FUNCTION_BLOCK FB_ROB_MANIP EXTENDS FB_ROB IMPLEMENTS ITF_2_6AxisRobot



VAR_OUTPUT

END_VAR
VAR

	tcppos, tcpvel : stPose3D;
	jointpos, jointvel: stJoint6;
	currFrame: stFrame;
	currTool: FB_Tool;

END_VAR

//State Machine

{warning 'Add method implementation '}
METHOD M_Home : BOOL
END_METHOD

{warning 'Add method implementation '}
METHOD M_SwitchTool : UINT
VAR_INPUT
	tool	: FB_Tool;
END_VAR
END_METHOD

{warning 'Add method implementation '}
METHOD MC_MoveAxesAbsolute : BOOL
VAR_INPUT
	target	: stTarget3D;
END_VAR
IF _state=eState.Active THEN
// 	P_TargetReached:=FALSE;
END_IF
END_METHOD

{warning 'Add method implementation '}
METHOD MC_MoveAxesRelative : BOOL
VAR_INPUT
	axes	: ARRAY [1..6] OF FB_Axis;
	offsets	: ARRAY [1..6] OF REAL;
END_VAR
END_METHOD

{warning 'Add method implementation '}
METHOD MC_MoveLinearAbsolute : BOOL
VAR_INPUT
	target	: stTarget3D;
END_VAR
END_METHOD

{warning 'Add method implementation '}
METHOD MC_ReadActualVelocity : stPose
END_METHOD

{warning 'Add method implementation '}
METHOD MC_ReadAnalogInput : LREAL
VAR_INPUT
	input	: INT;
END_VAR
END_METHOD

{warning 'Add method implementation '}
METHOD MC_ReadDigitalInput : BOOL
VAR_INPUT
	input	: INT;
END_VAR
END_METHOD

{warning 'Add method implementation '}
METHOD MC_SetDigitalOutput : BOOL
VAR_INPUT
	output	: INT;
	value	: BOOL;
END_VAR
END_METHOD

{warning 'Add method implementation '}
METHOD MC_SetOperationMode : BOOL
VAR_INPUT
	mode	: eMode;
END_VAR
_mode:=mode;
END_METHOD

METHOD onActivate : BOOL
// ---- Init ----
transitionresult:=eResult.None;



// ---- Change ----

// _mode:= eMode.Automatic;




// ---- Check ----
transitionresult := eResult.SUCCESS;


// ---- Change State ----
IF transitionresult= eResult.SUCCESS THEN
	P_State:=eState.Active;
ELSIF transitionresult= eResult.FAILURE THEN
	P_State:=eState.Inactive;
ELSIF transitionresult= eResult.ERROR THEN
	P_State:=eState.ErrorProcessing;
ELSE
	ADSLOGSTR(ADSLOG_MSGTYPE_WARN,'Transitionresult from onActivate is None','');
END_IF
END_METHOD

METHOD onCleanup : BOOL
// ---- Init ----
transitionresult:=eResult.None;



// ---- Change ----

_mode:= eMode.Manual;




// ---- Check ----
transitionresult := eResult.SUCCESS;


// ---- Change State ----
IF transitionresult= eResult.SUCCESS THEN
	P_State:=eState.Unconfigured;
ELSIF transitionresult= eResult.FAILURE THEN
	ADSLOGSTR(ADSLOG_MSGTYPE_WARN,'Transitionresult from onCleanup is FAILURE ','');
ELSIF transitionresult= eResult.ERROR THEN
	P_State:=eState.ErrorProcessing;
ELSE
	ADSLOGSTR(ADSLOG_MSGTYPE_WARN,'Transitionresult from onCleanup is NONE','');
END_IF
END_METHOD

METHOD onConfigure : BOOL
// ---- Init ----
transitionresult:=eResult.None;



// ---- Change ----

_mode:= eMode.Manual;




// ---- Check ----
transitionresult := eResult.SUCCESS;


// ---- Change State ----
IF transitionresult= eResult.SUCCESS THEN
	P_State:=eState.Inactive;
ELSIF transitionresult= eResult.FAILURE THEN
	P_State:=eState.Unconfigured;
ELSIF transitionresult= eResult.ERROR THEN
	P_State:=eState.ErrorProcessing;
ELSE
	ADSLOGSTR(ADSLOG_MSGTYPE_WARN,'Transitionresult from onConfigure is None','');
END_IF
END_METHOD

METHOD onDeactivate : BOOL
// ---- Init ----
transitionresult:=eResult.None;



// ---- Change ----

_mode:= eMode.Manual;




// ---- Check ----
transitionresult := eResult.SUCCESS;


// ---- Change State ----
IF transitionresult= eResult.SUCCESS THEN
	P_State:=eState.Inactive;
ELSIF transitionresult= eResult.FAILURE THEN
	ADSLOGSTR(ADSLOG_MSGTYPE_WARN,'Transitionresult from onDeactivate is FAILURE','');
ELSIF transitionresult= eResult.ERROR THEN
	P_State:=eState.ErrorProcessing;
ELSE
	ADSLOGSTR(ADSLOG_MSGTYPE_WARN,'Transitionresult from onDeactivate is None','');
END_IF
END_METHOD

METHOD onError : BOOL
// ---- Init ----
transitionresult:=eResult.None;



// ---- Change ----

_mode:= eMode.Manual;




// ---- Check ----
transitionresult := eResult.SUCCESS;


// ---- Change State ----
IF transitionresult= eResult.SUCCESS THEN
	P_State:=eState.Unconfigured;
ELSIF transitionresult= eResult.FAILURE THEN
	P_State:=eState.Finalized;
ELSIF transitionresult= eResult.ERROR THEN
	ADSLOGSTR(ADSLOG_MSGTYPE_WARN,'Transitionresult from onError is Error','');
ELSE
	ADSLOGSTR(ADSLOG_MSGTYPE_WARN,'Transitionresult from onError is None','');
END_IF
END_METHOD

METHOD onShutdown : BOOL
// ---- Init ----
transitionresult:=eResult.None;



// ---- Change ----

_mode:= eMode.Manual;




// ---- Check ----
transitionresult := eResult.SUCCESS;


// ---- Change State ----
IF transitionresult= eResult.SUCCESS THEN
	P_State:=eState.Finalized;
ELSIF transitionresult= eResult.FAILURE THEN
	ADSLOGSTR(ADSLOG_MSGTYPE_WARN,'Transitionresult from onShutdown is FAILURE','');
ELSIF transitionresult= eResult.ERROR THEN
	P_State:=eState.ErrorProcessing;
ELSE
	ADSLOGSTR(ADSLOG_MSGTYPE_WARN,'Transitionresult from onShutdown is None','');
END_IF
END_METHOD

{warning 'Add property implementation'}
PROPERTY P_ActualAxisPos : stJoint6
GET
P_ActualAxisPos:= jointpos;
END_GET
END_PROPERTY

{warning 'Add property implementation'}
PROPERTY P_ActualJointVelocity : stJoint6
GET
P_ActualJointVelocity:= jointvel;
END_GET
END_PROPERTY

{warning 'Add property implementation'}
PROPERTY P_ActualTCPPos : stPose3D
GET
P_ActualTCPPos:=tcppos;
END_GET
END_PROPERTY

{warning 'Add property implementation'}
PROPERTY P_ActualTCPVelocity : stPose3D
GET
P_ActualTCPVelocity:=tcpvel;
END_GET
END_PROPERTY

{warning 'Add property implementation'}
PROPERTY P_currentFrame : stFrame
GET
P_currentFrame := currFrame;
END_GET
SET
currFrame := P_currentFrame;
END_SET
END_PROPERTY

{warning 'Add property implementation'}
PROPERTY P_currentFrameID : UINT
GET
P_currentFrameID:= currFrame.frameId;
END_GET
END_PROPERTY

{warning 'Add property implementation'}
PROPERTY P_currentTool : FB_Tool
GET
P_currentTool:= currTool;
END_GET
SET
currTool:= P_currentTool;
END_SET
END_PROPERTY

{warning 'Add property implementation'}
PROPERTY P_IsInHomePosition : BOOL
GET
END_GET
END_PROPERTY

PROPERTY P_TargetReached : BOOL
GET
END_GET
END_PROPERTY

END_FUNCTION_BLOCK

(* stored: Version 1.1.0.1, ProductVersion 3.1.4026.18
   POU FB_ROB_MANIP: Id {21b924b4-0fb6-46ff-9fb7-f679235d19bb}, SpecialFunc None
   Folder MotionControl: Id {fc8c0aca-629b-4848-a20d-78e9ce6e9fda}
   Folder StateControl: Id {12a0430c-efeb-4d5c-9e24-8b660ff5f112}
   Method M_Home: Id {332921a2-9f70-499b-943d-00519405a468}
   Method M_SwitchTool: Id {8ccd8377-a0a9-4b8e-810b-34174cdec411}
   Method MC_MoveAxesAbsolute: Id {36f9f0d0-3360-4749-8362-ffb2170f0840}
   Method MC_MoveAxesRelative: Id {d4d7d377-1aa7-4fc3-9e59-f55d00fe8d35}
   Method MC_MoveLinearAbsolute: Id {af96fe73-c0fb-4331-8a41-58ccd3cdc293}
   Method MC_ReadActualVelocity: Id {e5d4eac9-56f1-4bad-8730-f186ead5097a}
   Method MC_ReadAnalogInput: Id {31640c85-0b1f-4824-a130-bbe550925ab2}
   Method MC_ReadDigitalInput: Id {31fdd754-1fe6-45cf-a4b2-d988dbb8460a}
   Method MC_SetDigitalOutput: Id {8ce879d8-c2db-4879-a4e0-e7565e752bef}
   Method MC_SetOperationMode: Id {4920400e-07f5-4ffe-a144-4f0f1bdf8f55}
   Method onActivate: Id {9316e65a-0316-4500-ae6c-6cb94521b4a3}
   Method onCleanup: Id {e5e12f85-b185-4c53-9b05-43d399837d67}
   Method onConfigure: Id {26716ca6-30dc-4ca6-8cda-d49a9720fe10}
   Method onDeactivate: Id {b783adc3-fff9-47d4-a61d-a6f66730c870}
   Method onError: Id {6305bb7b-0fb9-4e94-97bf-c149fc83cbee}
   Method onShutdown: Id {15a32cde-208f-43d2-8298-96af9abf0f63}
   Property P_ActualAxisPos: Id {c68b9d82-514b-4e83-b58e-69cf77564b19}
   Get Get: Id {2b353ef5-5db5-4268-89e1-d980ddc297fa}
   Property P_ActualJointVelocity: Id {947a6f2a-4f8a-49d4-9aa5-6819f46128db}
   Get Get: Id {bcb260e7-58e3-43cb-b050-6f35e444f22e}
   Property P_ActualTCPPos: Id {0ea3c3d9-9984-43b2-ac68-a1a8d409d11e}
   Get Get: Id {019c7e94-91db-4b36-9e6e-9be7d9fb51c3}
   Property P_ActualTCPVelocity: Id {cd04f35a-047d-478b-8cf7-b18ee8d2a4f9}
   Get Get: Id {c88b221c-0030-413b-abf3-a401e3f71088}
   Property P_currentFrame: Id {26c13a2e-22c9-42bf-93d2-6ec67f3d3b92}
   Get Get: Id {a653af18-d7cf-47f7-a4f7-cc2e6fc7b606}
   Set Set: Id {e6c6bc6d-2657-4d60-86e4-310cd9e6760e}
   Property P_currentFrameID: Id {1702473e-444c-4cd6-804e-8254e6795235}
   Get Get: Id {f7d65704-7385-4187-bf30-3f71423d6939}
   Property P_currentTool: Id {28bbf2d2-3b7d-40db-8479-5b32abdd2c79}
   Get Get: Id {53c5ea4e-aa4b-4197-b229-249acd63fd6c}
   Set Set: Id {3bc312a7-cdb2-4a49-8d8e-296c8b2ef79a}
   Property P_IsInHomePosition: Id {0f2fd807-aeed-459c-9c2b-f2325fe045e7}
   Get Get: Id {cc381350-4b9b-4a45-a9c1-b7537b47d8d7}
   Property P_TargetReached: Id {2d1820d4-8eb7-4322-8576-21d865cfd73c}
   Get Get: Id {1a88700a-2bd0-44c2-8984-ac880d8ae7d7} *)
